{attribute 'qualified_only'}
{attribute 'strict'}
{attribute 'to_string'}
TYPE E_Sample_LargeEnum : (
        None                      := 0,  (* No specific functionality assigned. *)
        ApparentPower             := 1,  (* Apparent power (VA). *)
        AQI                       := 2,  (* Air Quality Index (None). *)
        AtmosphericPressure       := 3,  (* Atmospheric pressure (Pa, hPa, bar). *)
        Battery                   := 4,  (* Battery level (%). *)
        BloodGlucoseConcentration := 5,  (* Blood glucose concentration (mg/dL, mmol/L). *)
        CarbonMonoxide            := 6,  (* Carbon Monoxide (ppm). *)
        CarbonDioxide             := 7,  (* Carbon Dioxide (ppm). *)
        Conductivity              := 8,  (* Conductivity (S/cm, mS/cm, µS/cm). *)
        Current                   := 9,  (* Electric current (A, mA). *)
        DataRate                  := 10, (* Data rate (bps, kbps, Mbps). *)
        DataSize                  := 11, (* Data size (bytes, MB, GB). *)
        Distance                  := 12, (* Distance (m, cm, mm). *)
        Duration                  := 13, (* Duration (s, ms, h). *)
        Energy                    := 14, (* Energy (Wh, kWh, J). *)
        EnergyStorage             := 15, (* Stored energy (Wh, kWh, J). *)
        Frequency                 := 16, (* Frequency (Hz, kHz). *)
        Gas                       := 17, (* Gas volume (m³, ft³). *)
        Humidity                  := 18, (* Humidity (%). *)
        Illuminance               := 19, (* Illuminance (lx). *)
        Irradiance                := 20, (* Irradiance (W/m²). *)
        Moisture                  := 21, (* Moisture (%). *)
        Monetary                  := 22, (* Monetary value (ISO4217 currency code). *)
        NitrogenDioxide           := 23, (* Nitrogen Dioxide (µg/m³). *)
        NitrogenMonoxide          := 24, (* Nitrogen Monoxide (µg/m³). *)
        NitrousOxide              := 25, (* Nitrous Oxide (µg/m³). *)
        Ozone                     := 26, (* Ozone concentration (µg/m³). *)
        PH                        := 27, (* Acidity/alkalinity (pH). *)
        PM1                       := 28, (* Particulate matter <= 1 μm (µg/m³). *)
        PM10                      := 29, (* Particulate matter <= 10 μm (µg/m³). *)
        PM25                      := 30, (* Particulate matter <= 2.5 μm (µg/m³). *)
        PowerFactor               := 31, (* Power factor (%). *)
        Power                     := 32, (* Power (W, kW). *)
        Precipitation             := 33, (* Precipitation (mm, in). *)
        PrecipitationIntensity    := 34, (* Precipitation intensity (mm/h, in/h). *)
        Pressure                  := 35, (* Pressure (Pa, hPa, bar, psi). *)
        ReactiveEnergy            := 36, (* Reactive energy (varh, kvarh, Mvarh). *)
        ReactivePower             := 37, (* Reactive power (var, kvar, Mvar). *)
        SignalStrength            := 38, (* Signal strength (dB, dBm). *)
        SoundPressure             := 39, (* Sound pressure (dB, dBA). *)
        Speed                     := 40, (* Speed (m/s, km/h, mph, kn). *)
        SulphurDioxide            := 41, (* Sulphur Dioxide (µg/m³). *)
        Temperature               := 42, (* Temperature (°C, °F, K). *)
        VolatileOrganicCompounds  := 43, (* Volatile Organic Compounds (µg/m³). *)
        Voltage                   := 44, (* Electric potential / voltage (V, mV). *)
        Volume                    := 45, (* Volume (L, mL, m³, gal). *)
        VolumeFlowRate            := 46, (* Volume flow rate (m³/h, L/min). *)
        Weight                    := 47, (* Weight (kg, g, mg, lb). *)
        WindSpeed                 := 48  (* Wind speed (m/s, km/h, mph, kn). *)
    );
END_TYPE

(* stored: Version 1.1.0.1, ProductVersion 3.1.4024.16
   DUT E_Sample_LargeEnum: Id {92e764cd-3e31-41ec-a0fa-1e0766bb84b3} *)
